// TIA Portal V18 export
// export: Created 2026-01-09T11:32:03.4844305Z, ExportSetting WithDefaults, DisplayName Totally Integrated Automation Portal, DisplayVersion V18 Update 5, DisplayName TIA Portal Openness, DisplayVersion V18 Update 5, DisplayName TIA Portal Teamcenter Gateway, DisplayVersion V18, DisplayName TIA Portal Version Control Interface, DisplayVersion V18, DisplayName SINAMICS Startdrive Advanced, DisplayVersion V18 SP2 Update 1, DisplayName SINAMICS Startdrive G110M, G120, G120C, G120D, G120P, G115D, DisplayVersion V18 SP2 Update 1, DisplayName SINAMICS Startdrive G130, G150, S120, S150, SINAMICS MV, S210, G220, S200, DisplayVersion V18 SP2 Update 1, DisplayName STEP 7 Professional, DisplayVersion V18 Update 5, DisplayName STEP 7 Safety, DisplayVersion V18, DisplayName WinCC Professional, DisplayVersion V18 Update 5
TagTable "ST_Com"
  ST_CommandRecord : Bool  (%DB[ST_SysDBNum].DBX50.3, CPU S71500-2PN_TP700, 1 s)
  ST_AutoRunningPause : Bool  (%DB[ST_SysDBNum].DBX100.2, CPU S71500-2PN_TP700, 1 s)
  ST_ScreenNo : Int  (%DB[ST_SysDBNum].DBW0, CPU S71500-2PN_TP700, 1 s)
    on ChangeValue: ActivateScreenByNumber(Screen number := , Object number := 0)
  ST_AutoRunning : Bool  (%DB[ST_SysDBNum].DBX100.1, CPU S71500-2PN_TP700, 1 s)
  ST_CommandTestLamp : Bool  (%DB[ST_SysDBNum].DBX50.4, CPU S71500-2PN_TP700, 1 s)
  ST_CommandBuzzerOn : Bool  (%DB[ST_SysDBNum].DBX50.5, CPU S71500-2PN_TP700, 1 s)
  ST_AutoRunningOver : Bool  (%DB[ST_SysDBNum].DBX100.3, CPU S71500-2PN_TP700, 1 s)
  ST_AutoStatus : Int  (%DB[ST_SysDBNum].DBW102, CPU S71500-2PN_TP700, 1 s)
  ST_CommandChangeOver : Bool  (%DB[ST_SysDBNum].DBX50.2, CPU S71500-2PN_TP700, 1 s)
  ST_StatusFinishProduct : DInt  (%DB[ST_SysDBNum].DBD16, CPU S71500-2PN_TP700, 1 s)
  ST_AlarmON : Bool  (%DB[ST_SysDBNum].DBX300.0, CPU S71500-2PN_TP700, 1 s)
  ST_SafetyLightCurtain[1] : Bool  (%DB[ST_SysDBNum].DBX200.1, CPU S71500-2PN_TP700, 1 s)
  ST_SafetyLightCurtain[0] : Bool  (%DB[ST_SysDBNum].DBX200.0, CPU S71500-2PN_TP700, 1 s)
  ST_SafetyLightCurtain[2] : Bool  (%DB[ST_SysDBNum].DBX200.2, CPU S71500-2PN_TP700, 1 s)
  ST_SafetyLightCurtain[3] : Bool  (%DB[ST_SysDBNum].DBX200.3, CPU S71500-2PN_TP700, 1 s)
  ST_SafetyLightCurtain[4] : Bool  (%DB[ST_SysDBNum].DBX200.4, CPU S71500-2PN_TP700, 1 s)
  ST_SafetyLightCurtain[5] : Bool  (%DB[ST_SysDBNum].DBX200.5, CPU S71500-2PN_TP700, 1 s)
  ST_SafetyLightCurtain[6] : Bool  (%DB[ST_SysDBNum].DBX200.6, CPU S71500-2PN_TP700, 1 s)
  ST_SafetyLightCurtain[7] : Bool  (%DB[ST_SysDBNum].DBX200.7, CPU S71500-2PN_TP700, 1 s)
  ST_SafetyDoorClose[0] : Bool  (%DB[ST_SysDBNum].DBX202.0, CPU S71500-2PN_TP700, 1 s)
  ST_SafetyDoorClose[1] : Bool  (%DB[ST_SysDBNum].DBX202.1, CPU S71500-2PN_TP700, 1 s)
  ST_SafetyDoorClose[2] : Bool  (%DB[ST_SysDBNum].DBX202.2, CPU S71500-2PN_TP700, 1 s)
  ST_SafetyDoorClose[3] : Bool  (%DB[ST_SysDBNum].DBX202.3, CPU S71500-2PN_TP700, 1 s)
  ST_SafetyDoorClose[4] : Bool  (%DB[ST_SysDBNum].DBX202.4, CPU S71500-2PN_TP700, 1 s)
  ST_SignalCheckSenor[1] : Bool  (%DB[ST_SysDBNum].DBX220.1, CPU S71500-2PN_TP700, 1 s)
  ST_SignalCheckSenor[2] : Bool  (%DB[ST_SysDBNum].DBX220.2, CPU S71500-2PN_TP700, 1 s)
  ST_SignalCheckSenor[3] : Bool  (%DB[ST_SysDBNum].DBX220.3, CPU S71500-2PN_TP700, 1 s)
  ST_SignalCheckSenor[4] : Bool  (%DB[ST_SysDBNum].DBX220.4, CPU S71500-2PN_TP700, 1 s)
  ST_UserName : String  (%DB[ST_SysDBNum].DBX700.0, CPU S71500-2PN_TP700, 1 s)
  ST_CommandOneCycle : Bool  (%DB[ST_SysDBNum].DBX51.2, CPU S71500-2PN_TP700, 1 s)
  ST_CommandDryRun : Bool  (%DB[ST_SysDBNum].DBX51.3, CPU S71500-2PN_TP700, 1 s)
  ST_CommandCalibration : Bool  (%DB[ST_SysDBNum].DBX51.4, CPU S71500-2PN_TP700, 1 s)
  ST_AlarmReset : Bool  (%DB[ST_SysDBNum].DBX300.2, CPU S71500-2PN_TP700, 1 s)
  ST10_Sys_Cmd_OnOffLine : Bool  (%DB[ST_SysDBNum].DBX51.1, CPU S71500-2PN_TP700, 1 s)
  ST_Start_Auto : Bool  (%DB[ST_SysDBNum].DBX100.6, CPU S71500-2PN_TP700, 1 s)
  ST_AllRun : Bool  (%DB[ST_SysDBNum].DBX100.7, CPU S71500-2PN_TP700, 1 s)
  ST_SysDBNum : Int  (1 s)   // Station sys DB No. / Číslo DB systému stanice
